{attribute 'GeneratedUsingTerminal: EL3443-0000-0016'}
{attribute addProperty BoxType "EL3443-0000-0016"}
{attribute addProperty Id "Voltage_Last_Zero_CrossingAT %I*ULINT8"}
{attribute addProperty CRC "3439292703"}
{attribute addProperty Size "8"}
TYPE L1_Timing_CCFF711F :
STRUCT
	{attribute addProperty Name "Voltage_Last_Zero_Crossing"}
	Voltage_Last_Zero_Crossing AT %I* : ULINT;
END_STRUCT
END_TYPE

(* stored: Version 1.2.0.0, ProductVersion 3.1.4024.9
   DUT L1_Timing_CCFF711F: Id {49550f10-f756-4113-bf2e-c255f1feecf3} *)
